FUNCTION_BLOCK OF_E_BLINK (* Simulates a blinking signal (turning on and off for specific durations) *)
  PACKAGE eclipse4diac::utils::signals;
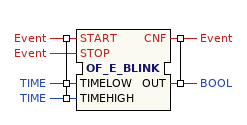
  EVENT_INPUT
    START WITH TIMELOW, TIMEHIGH; (* Start the perodic generation of events *)
    STOP; (* Stop the generation of events *)
  END_EVENT
  EVENT_OUTPUT
    CNF WITH OUT; (* Execution Confirmation *)
  END_EVENT
  VAR_INPUT
    TIMELOW : TIME; (* Time for OUT to be FALSE *)
    TIMEHIGH : TIME; (* Time for OUT to be TRUE *)
  END_VAR
  VAR_OUTPUT
    OUT : BOOL; (* Output value, starts with FALSE and switches between TRUE and FALSE for the given high and low times *)
  END_VAR
END_FUNCTION_BLOCK
